TYPE CurrentMeasurementStatuses :
STRUCT
	///Is the measurement valid?
	healthStatus: HealthStatus;
END_STRUCT
END_TYPE

(* stored: Version 1.1.0.1, ProductVersion 3.1.4019.2
   DUT CurrentMeasurementStatuses: Id {6c03c6d4-e3ff-44e1-af60-43ff15a9e93f} *)
